TYPE (* Package-qualified FORTE type name used during deployment *)
  (* Standard: 61499-1; Description: Copyright (c) 2026 Sichuan Qunyuan Technology Co., Ltd. This program and the accompanying materials are made available under the terms of the Eclipse Public License 2.0 which is available at https://www.eclipse.org/legal/epl-2.0/ SPDX-License-Identifier: EPL-2.0 *)
  (* Version 1.0, 2026-08-28, Zijun Tang, initial API and implementation *)
  PACKAGE eclipse4diac::core;
  {SET_ATTRIBUTE(TARGET, (IInterfaceElement:=FALSE,SubApp:=FALSE,FBType:=TRUE,Application:=FALSE,Connection:=FALSE,FB:=FALSE,DataType:=FALSE))}
  ForteTypeOverride : STRING := ''; (* FORTE type name for deployment (package-qualified or unqualified) *)
END_TYPE
